// TwinCAT 3 PLC project ModbusExt_Tests
// ProgramVersion: 3.1.4026.27
// libraries:
//   ModbusExt2, * (Beckhoff Automation)
//   Tc2_SerialCom, * (Beckhoff Automation GmbH)
//   Tc2_Standard, * (Beckhoff Automation GmbH)
//   Tc2_System, * (Beckhoff Automation GmbH)
// project tree:
//   / PlcTask.TcTTO
//   POUs/Test/ FB_Mb_TestBad.TcPOU, FB_Mb_TestGood.TcPOU, PRG_CodecTest.TcPOU, PRG_DeviceTest.TcPOU, PRG_LogWriterTest.TcPOU, PRG_RtuTest.TcPOU, PRG_TcpTest.TcPOU
// (motion and I/O tree: see PLC project modbusext2)
// real-time tasks:
//   TASK PlcTask1: cycle T#10ms, priority 21, ADS port 351
//   TASK PlcTask: cycle T#10ms, priority 20, ADS port 350

CONFIGURATION ModbusExt_Tests
    RESOURCE PLC ON TwinCAT3
        TASK PlcTask(INTERVAL := T#10ms, PRIORITY := 21);
        PROGRAM PRG_CodecTest WITH PlcTask : PRG_CodecTest;
        PROGRAM PRG_DeviceTest WITH PlcTask : PRG_DeviceTest;
        PROGRAM PRG_LogWriterTest WITH PlcTask : PRG_LogWriterTest;
        PROGRAM PRG_RtuTest WITH PlcTask : PRG_RtuTest;
        PROGRAM PRG_TcpTest WITH PlcTask : PRG_TcpTest;
    END_RESOURCE
END_CONFIGURATION

// ---- POUs/Test/PRG_CodecTest.TcPOU
PROGRAM PRG_CodecTest
VAR
	bRun            : BOOL := TRUE;     // Set TRUE online to re-run
	bAllPass        : BOOL;

	bCrcPass        : BOOL;
	bBuildPass      : BOOL;
	bParsePass      : BOOL;
	bExceptionPass  : BOOL;
	bMalformedPass  : BOOL;
	bTruncatedPass  : BOOL;

	wCrc            : WORD;
	nLen            : UINT;
	bOk             : BOOL;
	stRes           : ST_MbParseResult;
	aPdu            : ARRAY[0..259] OF BYTE;

	// Spec example: read 3 holding registers from unit 16#11 starting at 40108
	aFrame          : ARRAY[0..5] OF BYTE := [16#11, 16#03, 16#00, 16#6B, 16#00, 16#03];
	aResp           : ARRAY[0..7] OF BYTE := [16#03, 16#06, 16#AE, 16#41, 16#56, 16#52, 16#43, 16#40];
	aExc            : ARRAY[0..1] OF BYTE := [16#83, 16#02];
	aBad            : ARRAY[0..7] OF BYTE := [16#03, 16#04, 16#AE, 16#41, 16#56, 16#52, 16#43, 16#40];
END_VAR

IF NOT bRun THEN
	RETURN;
END_IF
bRun := FALSE;

// 1. CRC over 11 03 00 6B 00 03 -> 16#8776 (wire order 76 87)
wCrc := F_MbCrc16(ADR(aFrame), SIZEOF(aFrame));
bCrcPass := (wCrc = 16#8776);

// 2. Build FC3, offset 16#6B, qty 3 -> 03 00 6B 00 03
F_MbMemSet(ADR(aPdu), 0, SIZEOF(aPdu));
nLen := F_MbBuildRequest(GVL_MbConst.FC_READ_HOLDING, 16#6B, 3, 0, 0, ADR(aPdu), SIZEOF(aPdu));
bBuildPass := (nLen = 5) AND (aPdu[0] = 16#03) AND (aPdu[1] = 16#00) AND (aPdu[2] = 16#6B)
              AND (aPdu[3] = 16#00) AND (aPdu[4] = 16#03);

// 3. Good FC3 response, 3 registers
bOk := F_MbParseResponse(ADR(aResp), SIZEOF(aResp), GVL_MbConst.FC_READ_HOLDING, 3, stRes);
bParsePass := bOk AND stRes.bOk AND (stRes.nByteCount = 6) AND (stRes.nDataOffset = 2)
              AND (stRes.eClass = E_MbErrorClass.None);

// 4. Exception 83 02
bOk := F_MbParseResponse(ADR(aExc), SIZEOF(aExc), GVL_MbConst.FC_READ_HOLDING, 3, stRes);
bExceptionPass := (NOT bOk) AND stRes.bException AND (stRes.nExcCode = 2)
                  AND (stRes.eClass = E_MbErrorClass.Exception);

// 5. Byte count disagrees with quantity
bOk := F_MbParseResponse(ADR(aBad), SIZEOF(aBad), GVL_MbConst.FC_READ_HOLDING, 3, stRes);
bMalformedPass := (NOT bOk) AND (stRes.eClass = E_MbErrorClass.Malformed);

// 6. Short frame
bOk := F_MbParseResponse(ADR(aResp), 4, GVL_MbConst.FC_READ_HOLDING, 3, stRes);
bTruncatedPass := (NOT bOk) AND (stRes.eClass = E_MbErrorClass.Truncated);

bAllPass := bCrcPass AND bBuildPass AND bParsePass AND bExceptionPass AND bMalformedPass AND bTruncatedPass;

END_PROGRAM

// ---- POUs/Test/PRG_DeviceTest.TcPOU
PROGRAM PRG_DeviceTest
VAR
	fbMock         : FB_MbTransportMock;
	fbGood         : FB_Mb_TestGood;
	fbBad          : FB_Mb_TestBad;
	stLogGood      : ST_MbLog;
	stLogBad       : ST_MbLog;
	fbExport	   : FB_MbLogExport;
	
	fbGood2   : FB_Mb_TestGood;
	stLogGood2 : ST_MbLog;
	nReqLast  : UDINT;
	nReq1     : UDINT;
	nReq2     : UDINT;
	bArbPass  : BOOL;

	bMemInit       : BOOL;
	bGoodPass      : BOOL;
	bBadPass       : BOOL;
	bSplitPass     : BOOL;
	bReadPass      : BOOL;
	bWritePass     : BOOL;
	bHandshakePass : BOOL;
	bOnlineChangePass : BOOL;
	nWriteStep     : UINT;
	bExport		   : BOOL;
END_VAR

IF NOT bMemInit THEN
	bMemInit := TRUE;
	fbMock.aHolding[0]   := 1234;
	fbMock.aHolding[1]   := 500;                                        // Hr2: 0..1000 -> 0..100 = 50.0
	fbMock.aHolding[2]   := 16#0000; fbMock.aHolding[3]   := 16#3FC0;   // Hr3: 1.5 REAL, CDAB
	fbMock.aHolding[9]   := 16#86A0; fbMock.aHolding[10]  := 16#0001;   // Hr4: 100000 UDINT, CDAB
	fbMock.aHolding[99]  := 16#4D6F; fbMock.aHolding[100] := 16#6462;   // Hr5: 'ModbusExt'
	fbMock.aHolding[101] := 16#7573; fbMock.aHolding[102] := 16#4578;
	fbMock.aHolding[103] := 16#7400;
	fbMock.aHolding[115] := 42;                                         // Hr6 (slow)
	fbMock.aHolding[299] := 16#0008;                                    // Status bit 3
	fbMock.aInput[0]     := 16#0000; fbMock.aInput[1]     := 16#4020;   // Ir1: 2.5
	fbMock.aInput[2]     := 7;       fbMock.aInput[3]     := 0;         // Ir2: 7
	fbMock.aCoils[0]     := TRUE;    fbMock.aCoils[1]     := FALSE;
	fbMock.aDiscrete[0]  := TRUE;
	fbMock.bExcOnRange   := TRUE;
	fbMock.nExcOffset    := 5;                                          // Undefined register inside the first HR block's gap
END_IF

fbMock.aHolding[399] := 55;
fbMock.aHolding[409] := 56;
fbMock.aHolding[419] := 57;

fbGood(itfTransport := fbMock, bEnable := TRUE, refLog := stLogGood);
fbBad(bEnable := TRUE, refLog := stLogBad, bLogToFile := FALSE);

fbGood2(itfTransport := fbMock, nUnitId := 2, bEnable := TRUE, refLog := stLogGood2);

// Attribute each mock request to the unit that sent it
IF fbMock.nRequests <> nReqLast THEN
	nReqLast := fbMock.nRequests;
	IF fbMock.nLastUnit = 1 THEN
		nReq1 := nReq1 + 1;
	ELSIF fbMock.nLastUnit = 2 THEN
		nReq2 := nReq2 + 1;
	END_IF
END_IF

// Both online, both reading, and the bus split roughly evenly
bArbPass := fbGood2.bOnline AND fbGood2.Hr1.bValid AND fbGood2.Ir1.bValid
            AND (nReq1 > 50) AND (nReq2 > 50)
            AND (nReq2 > nReq1 / 2) AND (nReq1 > nReq2 / 2);

// Config
bGoodPass  := (NOT fbGood.bConfigError) AND (fbGood.nPoints = 16);
bBadPass   := fbBad.bConfigError AND (fbBad.nBlocks = 0) AND (stLogBad.nCount = 7);

// Self-split: 7 blocks -> 9, first two log entries are the two exceptions
bSplitPass := (fbGood.nBlocks = 12)
              AND (stLogGood.aEntries[0].eClass = E_MbErrorClass.Exception)
              AND (stLogGood.aEntries[1].eClass = E_MbErrorClass.Exception);

bOnlineChangePass := fbGood.Hr8.bValid AND (fbGood.Hr8.fValue = 55) AND (fbGood.Hr1.fValue = 777);
			  
// Reads (latched: the writes below change Hr1/Hr2/Hr3/Coil2 afterwards)
bReadPass := bReadPass OR (fbGood.bOnline
	AND fbGood.Hr1.bValid AND (fbGood.Hr1.fValue = 1234)
	AND (fbGood.Hr2.fValue = 50.0)
	AND (fbGood.Hr3.fValue = 1.5)
	AND (fbGood.Hr4.fValue = 100000)
	AND (fbGood.Hr5.sValue = 'ModbusExt')
	AND fbGood.Hr6.bValid AND (fbGood.Hr6.fValue = 42)
	AND (fbGood.Status.fValue = 1)
	AND (fbGood.Ir1.fValue = 2.5) AND (fbGood.Ir2.fValue = 7)
	AND (fbGood.Coil1.fValue = 1) AND fbGood.Coil2.bValid AND (fbGood.Coil2.fValue = 0)
	AND (fbGood.Di1.fValue = 1)
	AND (NOT fbGood.Hr7.bValid));

// Writes
CASE nWriteStep OF
	0:
		IF bReadPass THEN
			fbGood.Hr1.fWriteValue   := 777;   fbGood.Hr1.bWriteReq   := TRUE;
			fbGood.Hr2.fWriteValue   := 25.0;  fbGood.Hr2.bWriteReq   := TRUE;   // eng 25 -> raw 250
			fbGood.Hr3.fWriteValue   := 3.25;  fbGood.Hr3.bWriteReq   := TRUE;   // REAL, CDAB
			fbGood.Coil2.fWriteValue := 1;     fbGood.Coil2.bWriteReq := TRUE;
			fbGood.Ir1.fWriteValue   := 1;     fbGood.Ir1.bWriteReq   := TRUE;   // read-only -> Err
			fbGood.Hr4.fWriteValue   := 5.0E9; fbGood.Hr4.bWriteReq   := TRUE;   // beyond UInt32 -> Err
			nWriteStep := 1;
		END_IF
	1:
		IF fbGood.Hr1.bWriteDone AND fbGood.Hr2.bWriteDone AND fbGood.Hr3.bWriteDone AND fbGood.Coil2.bWriteDone
		   AND fbGood.Ir1.bWriteErr AND fbGood.Hr4.bWriteErr THEN
			bWritePass := (fbMock.aHolding[0] = 777) AND (fbMock.aHolding[1] = 250)
			              AND (fbMock.aHolding[2] = 16#0000) AND (fbMock.aHolding[3] = 16#4050)
			              AND fbMock.aCoils[1];
			fbGood.Hr1.bWriteReq   := FALSE;
			fbGood.Hr2.bWriteReq   := FALSE;
			fbGood.Hr3.bWriteReq   := FALSE;
			fbGood.Coil2.bWriteReq := FALSE;
			fbGood.Ir1.bWriteReq   := FALSE;
			fbGood.Hr4.bWriteReq   := FALSE;
			nWriteStep := 2;
		END_IF
	2:
		IF (NOT fbGood.Hr1.bWriteDone) AND (NOT fbGood.Ir1.bWriteErr) AND (NOT fbGood.Hr1.bWriteBusy)
		   AND (fbGood.Hr1.fValue = 777) AND (fbGood.Hr3.fValue = 3.25) AND (fbGood.Coil2.fValue = 1) THEN
			bHandshakePass := TRUE;
			nWriteStep := 3;
		END_IF
END_CASE

fbExport(sPath := 'C:\ModbusExt\TestGood.csv', bExecute := bExport, refLog := stLogGood);

END_PROGRAM

// ---- POUs/Test/FB_Mb_TestGood.TcPOU
FUNCTION_BLOCK FB_Mb_TestGood EXTENDS FB_ModbusDevice
VAR_INPUT
	// Holding registers: 40001..40004 contiguous, 40010 within gap 8 -> one block
	Hr1    : ST_MbPoint := (nAddr := 40001);
	Hr2    : ST_MbPoint := (nAddr := 40002, eType := E_MbType.Int16, fRawMin := 0, fRawMax := 1000, fEngMin := 0, fEngMax := 100);
	Hr3    : ST_MbPoint := (nAddr := 40003, eType := E_MbType.Real32);
	Hr4    : ST_MbPoint := (nAddr := 40010, eType := E_MbType.UInt32);
	// Gap > 8 -> second block
	Hr5    : ST_MbPoint := (nAddr := 40100, eType := E_MbType.Text, nRegs := 8);
	// Slow -> its own block
	Hr6    : ST_MbPoint := (nAddr := 40116, ePoll := E_MbPoll.Slow);
	// Off -> no block
	Hr7    : ST_MbPoint := (nAddr := 40200, ePoll := E_MbPoll.Off);
	// Far away -> third fast HR block
	Hr8    : ST_MbPoint := (nAddr := 40400);
	Hr9    : ST_MbPoint := (nAddr := 40410);
	Hr10   : ST_MbPoint := (nAddr := 40420);
	Status : ST_MbPoint := (nAddr := 40300, eType := E_MbType.RegisterBit, nBit := 3);
	// Input registers, contiguous -> one block
	Ir1    : ST_MbPoint := (nAddr := 30001, eType := E_MbType.Real32);
	Ir2    : ST_MbPoint := (nAddr := 30003, eType := E_MbType.UInt32);
	// Coils and a discrete input
	Coil1  : ST_MbPoint := (nAddr := 1);
	Coil2  : ST_MbPoint := (nAddr := 2);
	Di1    : ST_MbPoint := (nAddr := 10001);
END_VAR

Register();
SUPER^();

//FB_Init is always available implicitly and it is used primarily for initialization.
//The return value is not evaluated. For a specific influence, you can also declare the
//methods explicitly and provide additional code there with the standard initialization
//code. You can evaluate the return value.
METHOD FB_Init: BOOL
VAR_INPUT
    bInitRetains: BOOL; // TRUE: the retain variables are initialized (reset warm / reset cold)
    bInCopyCode: BOOL;  // TRUE: the instance will be copied to the copy code afterward (online change)   
END_VAR
Register();
END_METHOD

METHOD FB_Reinit: BOOL
VAR_INPUT   
END_VAR
Register();
END_METHOD

METHOD PRIVATE Register
Profile(sModel := 'TestGood', eWordOrder := E_MbWordOrder.CDAB);
AddPoint(Hr1, 'Hr1');
AddPoint(Hr2, 'Hr2');
AddPoint(Hr3, 'Hr3');
AddPoint(Hr4, 'Hr4');
AddPoint(Hr5, 'Hr5');
AddPoint(Hr6, 'Hr6');
AddPoint(Hr7, 'Hr7');
AddPoint(Hr8, 'Hr8');
AddPoint(Hr9, 'Hr9');
AddPoint(Hr10, 'Hr10');
AddPoint(Status, 'Status');
AddPoint(Ir1, 'Ir1');
AddPoint(Ir2, 'Ir2');
AddPoint(Coil1, 'Coil1');
AddPoint(Coil2, 'Coil2');
AddPoint(Di1, 'Di1');
END_METHOD

END_FUNCTION_BLOCK

// ---- POUs/Test/FB_Mb_TestBad.TcPOU
FUNCTION_BLOCK FB_Mb_TestBad EXTENDS FB_ModbusDevice
VAR_INPUT
	A : ST_MbPoint := (nAddr := 40001);
	B : ST_MbPoint := (nAddr := 40001);                                               // overlap + duplicate name
	C : ST_MbPoint := (nAddr := 20005);                                               // no Modicon range
	D : ST_MbPoint := (nAddr := 40010, eType := E_MbType.RegisterBit, nBit := 16);   // bit out of range
	E : ST_MbPoint := (nAddr := 40020, fEngMax := 100);                               // eng range without raw range
	F : ST_MbPoint := (nAddr := 40030, eType := E_MbType.Text);                       // nRegs missing
	G : ST_MbPoint := (nAddr := 10001, eType := E_MbType.Int16);                      // integer type on a bit region
END_VAR

Register();
SUPER^();

//FB_Init is always available implicitly and it is used primarily for initialization.
//The return value is not evaluated. For a specific influence, you can also declare the
//methods explicitly and provide additional code there with the standard initialization
//code. You can evaluate the return value.
METHOD FB_Init: BOOL
VAR_INPUT
    bInitRetains: BOOL; // TRUE: the retain variables are initialized (reset warm / reset cold)
    bInCopyCode: BOOL;  // TRUE: the instance will be copied to the copy code afterward (online change)   
END_VAR
Register();
END_METHOD

METHOD FB_Reinit: BOOL
VAR_INPUT   
END_VAR
Register();
END_METHOD

METHOD Register
Profile(sModel := 'TestBad');
AddPoint(A, 'A');
AddPoint(B, 'A');
AddPoint(C, 'C');
AddPoint(D, 'D');
AddPoint(E, 'E');
AddPoint(F, 'F');
AddPoint(G, 'G');
END_METHOD

END_FUNCTION_BLOCK

// ---- POUs/Test/PRG_LogWriterTest.TcPOU
PROGRAM PRG_LogWriterTest
VAR
	fbWriter  : FB_MbLogWriter;
	stLog     : ST_MbLog;
	fbSysTime : GETSYSTEMTIME;
	tNow      : ULINT;
	bAddOne   : BOOL;          // Set online: appends one entry to the ring
	bAddBurst : BOOL;          // Set online: appends 150 entries at once (exceeds the ring)
	nCount    : UDINT;
	i         : UINT;
END_VAR

fbSysTime();
tNow := SHL(DWORD_TO_ULINT(fbSysTime.timeHiDW), 32) + DWORD_TO_ULINT(fbSysTime.timeLoDW);

IF bAddOne THEN
	bAddOne := FALSE;
	Append();
END_IF
IF bAddBurst THEN
	bAddBurst := FALSE;
	FOR i := 1 TO 150 DO
		Append();
	END_FOR
END_IF

fbWriter(sDir := 'C:\ModbusExt\Logs', sName := 'WriterTest', pLog := ADR(stLog), tNow := tNow);

METHOD Append
nCount := nCount + 1;
stLog.aEntries[stLog.nHead].tTime    := tNow;
stLog.aEntries[stLog.nHead].sName    := CONCAT('Entry', UDINT_TO_STRING(nCount));
stLog.aEntries[stLog.nHead].nUnitId  := 1;
stLog.aEntries[stLog.nHead].eRegion  := E_MbRegion.HoldingRegister;
stLog.aEntries[stLog.nHead].nAddr    := 40000 + nCount;
stLog.aEntries[stLog.nHead].nFc      := 3;
stLog.aEntries[stLog.nHead].eOp      := E_MbOp.Read;
stLog.aEntries[stLog.nHead].eClass   := E_MbErrorClass.Timeout;
stLog.nHead := (stLog.nHead + 1) MOD GVL_MbParam.MB_LOG_SIZE;
IF stLog.nCount < GVL_MbParam.MB_LOG_SIZE THEN stLog.nCount := stLog.nCount + 1; END_IF
stLog.nSeq := stLog.nSeq + 1;
END_METHOD

END_PROGRAM

// ---- POUs/Test/PRG_RtuTest.TcPOU
PROGRAM PRG_RtuTest
VAR
	stEl6In1  AT %I* : EL6inData22B;
	stEl6Out1 AT %Q* : EL6outData22B;
	fbRs485   : FB_MbTransportRtu;
	fbDev     : FB_Mb_TestGood;
	stLog     : ST_MbLog;
END_VAR

fbRs485(pComIn := ADR(stEl6In1), pComOut := ADR(stEl6Out1), nSizeComIn := SIZEOF(stEl6In1));
fbDev(itfTransport := fbRs485, nUnitId := 1, bEnable := TRUE, refLog := stLog);

END_PROGRAM

// ---- POUs/Test/PRG_TcpTest.TcPOU
PROGRAM PRG_TcpTest
VAR
	fbTcp    : FB_MbTransportTcp := (sHost := '127.0.0.1', nPort := 502);
	fbDev    : FB_Mb_TestGood;
	stLog    : ST_MbLog;
	bTcpPass : BOOL;
END_VAR

fbTcp();
fbDev(itfTransport := fbTcp, nUnitId := 1, bEnable := TRUE, refLog := stLog);

bTcpPass := fbTcp.bConnected AND fbDev.bOnline
            AND (fbDev.Hr1.fValue = 1234) AND (fbDev.Hr2.fValue = 50.0) AND (fbDev.Hr3.fValue = 1.5);

END_PROGRAM
